(* IEC 61131-3 sources: esstee/src/tests/programs/function, 9 files *)

(* ---- badinput.ST ---- *)
FUNCTION my_func : INT

VAR
	not_in : INT;
END_VAR

VAR_INPUT
	in1 : INT;
	in2 : INT;
END_VAR

;

END_FUNCTION

PROGRAM t

VAR
	a : INT;
	b : INT;
	c : INT;
	d : INT;
END_VAR

c := my_func("wrong_type", in2:=false);

END_PROGRAM

(* ---- badinputname.ST ---- *)
FUNCTION my_func : INT

VAR
	not_in : INT;
END_VAR

VAR_INPUT
	in1 : INT;
	in2 : INT;
END_VAR

;

END_FUNCTION

PROGRAM t

VAR
	a : INT;
	b : INT;
	c : INT;
	d : INT;
END_VAR

c := my_func(bad=1);

END_PROGRAM

(* ---- badnotin.ST ---- *)
FUNCTION my_func : INT

VAR
	not_in : INT;
END_VAR

VAR_INPUT
	in1 : INT;
	in2 : INT;
END_VAR

;

END_FUNCTION

PROGRAM t

VAR
	a : INT;
	b : INT;
	c : INT;
	d : INT;
END_VAR

c := my_func(not_in:=1);

END_PROGRAM

(* ---- badtoomany.ST ---- *)
FUNCTION my_func : INT

VAR
	not_in : INT;
END_VAR

VAR_INPUT
	in1 : INT;
	in2 : INT;
END_VAR

;

END_FUNCTION

PROGRAM t

VAR
	a : INT;
	b : INT;
	c : INT;
	d : INT;
END_VAR

c := my_func(1, 2, 3);

END_PROGRAM

(* ---- disjointin.ST ---- *)
FUNCTION my_func : INT

VAR
	not_in : INT;
END_VAR

VAR_INPUT
	in1 : INT;
END_VAR

VAR
	a : INT;
END_VAR

VAR_INPUT
	in2 : INT;
END_VAR

my_func := in1 - in2;

END_FUNCTION

PROGRAM t

VAR
	a : INT;
	b : INT;
	c : INT;
	d : INT;
END_VAR

c := my_func(a,b);

d := my_func(in1:=a,in2:=b);

END_PROGRAM

(* ---- funcparams.ST ---- *)
FUNCTION my_func : INT

VAR_INPUT
	in1 : INT;
	in2 : INT;
END_VAR

my_func := in1 + in2;

END_FUNCTION

PROGRAM t

VAR
	a : INT;
	b : INT;
	c : INT;
	d : INT;
END_VAR

c := my_func(1+1, my_func(4*10, 5));

d := my_func(a, a*10);

END_PROGRAM

(* ---- min.ST ---- *)
FUNCTION my_min : INT

VAR_INPUT
	val1 : INT;
	val2 : INT;
END_VAR

if val1 < val2 then
   my_min := val1;
else
   my_min := val2;
end_if;

END_FUNCTION

PROGRAM t

VAR
	a : INT;
	b : INT;
	c : INT;
	d : INT;
END_VAR

c := my_min(a, b);

d := my_min(b, a);

END_PROGRAM

(* ---- recursion.ST ---- *)
FUNCTION my_func : INT

VAR_INPUT
	in1 : INT;
	in2 : INT;
END_VAR

my_func := in1 + in2;

END_FUNCTION

PROGRAM t

VAR
	a : INT;
	b : INT;
	c : INT;
	d : INT;
END_VAR

c := my_func(my_func(4,5),1+1);

d := my_func(a, 10*a);

END_PROGRAM

(* ---- reset.ST ---- *)
FUNCTION my_func : INT

VAR
	not_in : INT;
END_VAR

VAR_INPUT
	in1 : INT;
	in2 : INT;
END_VAR

my_func := in1 + in2;

END_FUNCTION

PROGRAM t

VAR
	a : INT;
	b : INT;
	c : INT;
	d : INT;
END_VAR

c := my_func(10,20);

d := my_func();

END_PROGRAM
